FUNCTION F_ResetCircuitBreakerGlobals : BOOL
VAR_INPUT
END_VAR
VAR
END_VAR

GVL_Logger.bTrickleTripped := FALSE;
GVL_Logger.nGlobAccEvents := 0;

END_FUNCTION

(* stored: Version 1.1.0.1
   POU F_ResetCircuitBreakerGlobals: Id {af07064f-81b8-4e8e-bacc-84cfa4b1f877}, SpecialFunc None *)
